PROGRAM MAIN
VAR
END_VAR

PRG_DIAGNOSTIC();
PRG_GATT();

END_PROGRAM

(* stored: Version 1.1.0.1, ProductVersion 3.1.4022.12
   POU MAIN: Id {9423868c-bdb9-4247-bc56-5f1baa6fbd52}, SpecialFunc None *)
